// Mitsubishi GX Works2 project: PLC-Servo 실습 과제 1   PLC: Q03UDV

PROGRAM MAIN
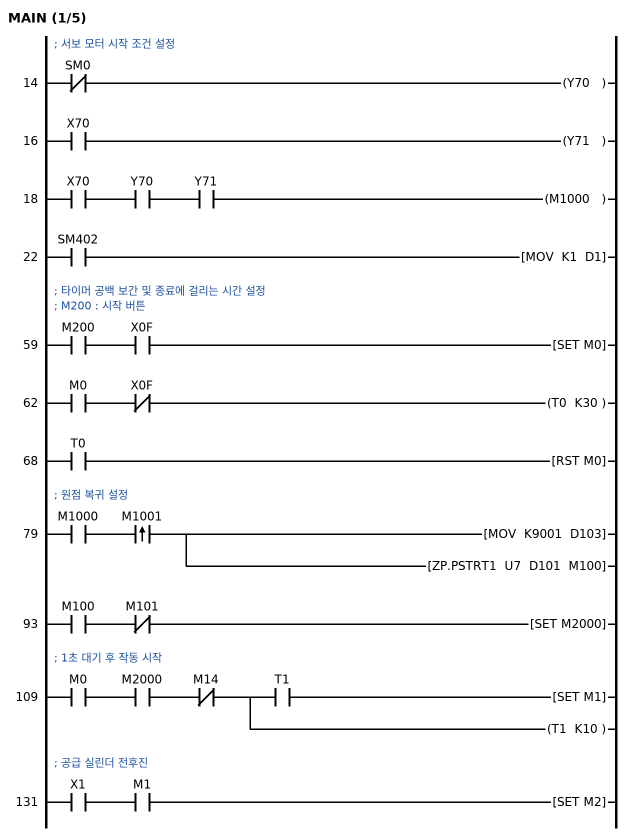
; 서보 모터 시작 조건 설정
14    LDI     SM0
      OUT     Y70
16    LD      X70
      OUT     Y71
18    LD      X70
      AND     Y70
      AND     Y71
      OUT     M1000
22    LD      SM402
      MOV     K1 D1
; 타이머 공백 보간 및 종료에 걸리는 시간 설정
; M200 : 시작 버튼
59    LD      M200
      AND     X0F
      SET     M0
62    LD      M0
      ANI     X0F
      OUT     T0 K30
68    LD      T0
      RST     M0
; 원점 복귀 설정
79    LD      M1000
      ANDP    M1001
      MOV     K9001 D103
      ZP.PSTRT1 U7 D101 M100
93    LD      M100
      ANI     M101
      SET     M2000
; 1초 대기 후 작동 시작
109   LD      M0
      AND     M2000
      ANI     M14
      MPS
      AND     T1
      SET     M1
      MPP
      OUT     T1 K10
; 공급 실린더 전후진
131   LD      X1
      AND     M1
      SET     M2
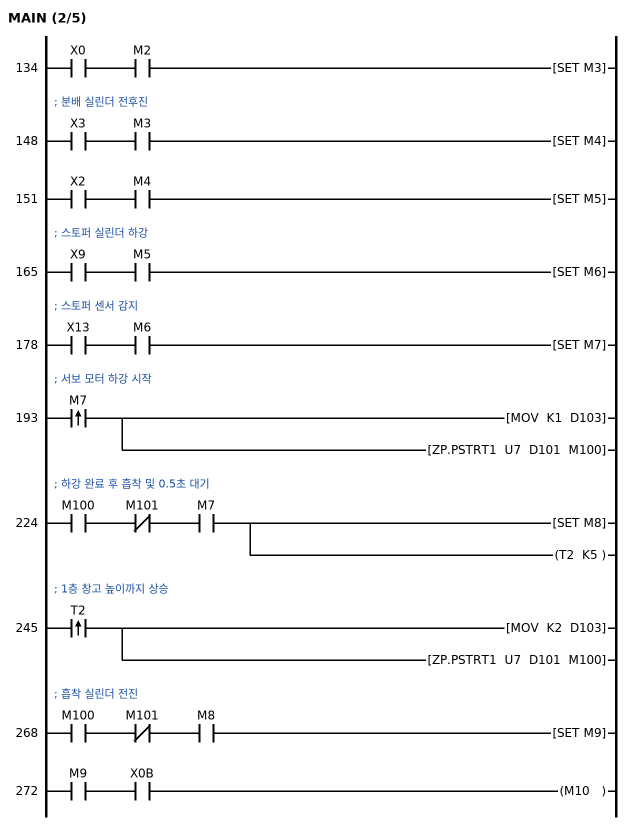
134   LD      X0
      AND     M2
      SET     M3
; 분배 실린더 전후진
148   LD      X3
      AND     M3
      SET     M4
151   LD      X2
      AND     M4
      SET     M5
; 스토퍼 실린더 하강
165   LD      X9
      AND     M5
      SET     M6
; 스토퍼 센서 감지
178   LD      X13
      AND     M6
      SET     M7
; 서보 모터 하강 시작
193   LDP     M7
      MOV     K1 D103
      ZP.PSTRT1 U7 D101 M100
; 하강 완료 후 흡착 및 0.5초 대기
224   LD      M100
      ANI     M101
      AND     M7
      SET     M8
      OUT     T2 K5
; 1층 창고 높이까지 상승
245   LDP     T2
      MOV     K2 D103
      ZP.PSTRT1 U7 D101 M100
; 흡착 실린더 전진
268   LD      M100
      ANI     M101
      AND     M8
      SET     M9
272   LD      M9
      AND     X0B
      OUT     M10
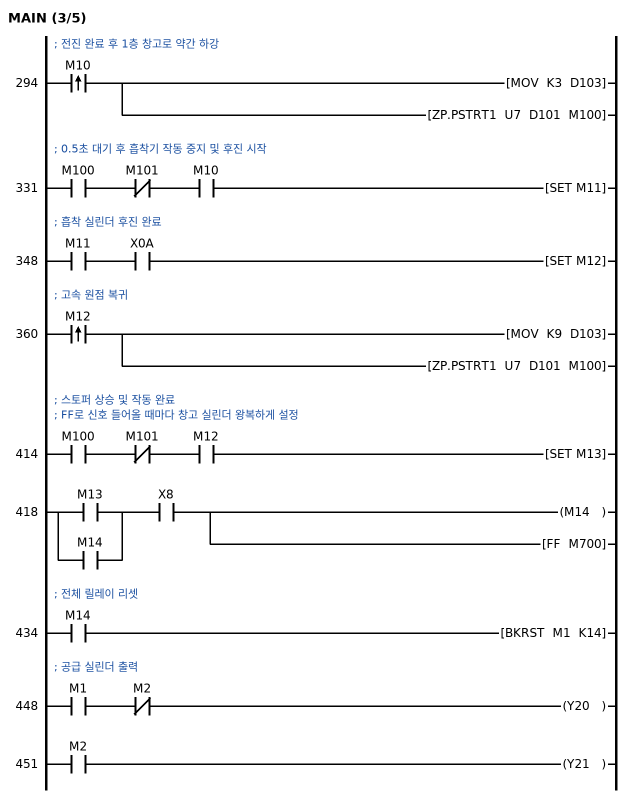
; 전진 완료 후 1층 창고로 약간 하강
294   LDP     M10
      MOV     K3 D103
      ZP.PSTRT1 U7 D101 M100
; 0.5초 대기 후 흡착기 작동 중지 및 후진 시작
331   LD      M100
      ANI     M101
      AND     M10
      SET     M11
; 흡착 실린더 후진 완료
348   LD      M11
      AND     X0A
      SET     M12
; 고속 원점 복귀
360   LDP     M12
      MOV     K9 D103
      ZP.PSTRT1 U7 D101 M100
; 스토퍼 상승 및 작동 완료
; FF로 신호 들어올 때마다 창고 실린더 왕복하게 설정
414   LD      M100
      ANI     M101
      AND     M12
      SET     M13
418   LD      M13
      OR      M14
      AND     X8
      OUT     M14
      FF      M700
; 전체 릴레이 리셋
434   LD      M14
      BKRST   M1 K14
; 공급 실린더 출력
448   LD      M1
      ANI     M2
      OUT     Y20
451   LD      M2
      OUT     Y21
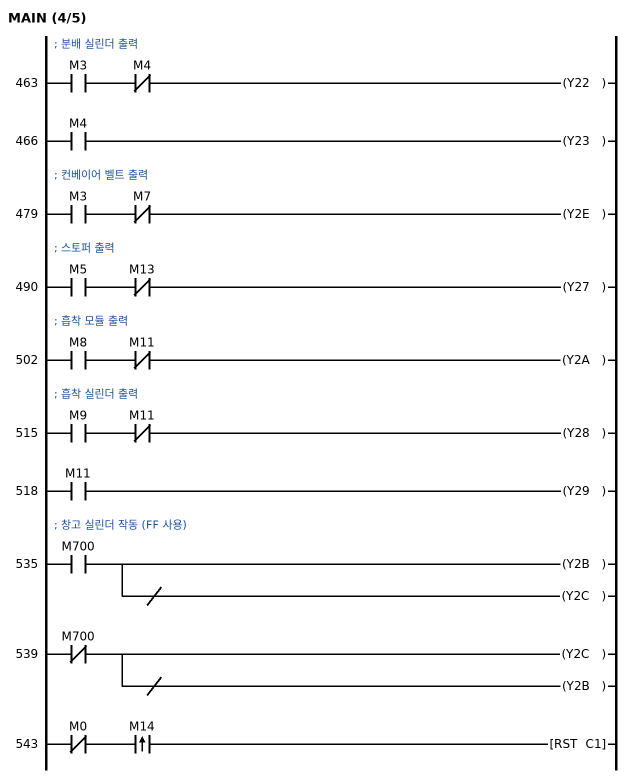
; 분배 실린더 출력
463   LD      M3
      ANI     M4
      OUT     Y22
466   LD      M4
      OUT     Y23
; 컨베이어 벨트 출력
479   LD      M3
      ANI     M7
      OUT     Y2E
; 스토퍼 출력
490   LD      M5
      ANI     M13
      OUT     Y27
; 흡착 모듈 출력
502   LD      M8
      ANI     M11
      OUT     Y2A
; 흡착 실린더 출력
515   LD      M9
      ANI     M11
      OUT     Y28
518   LD      M11
      OUT     Y29
; 창고 실린더 작동 (FF 사용)
535   LD      M700
      OUT     Y2B
      INV
      OUT     Y2C
539   LDI     M700
      OUT     Y2C
      INV
      OUT     Y2B
543   LDI     M0
      ANDP    M14
      RST     C1
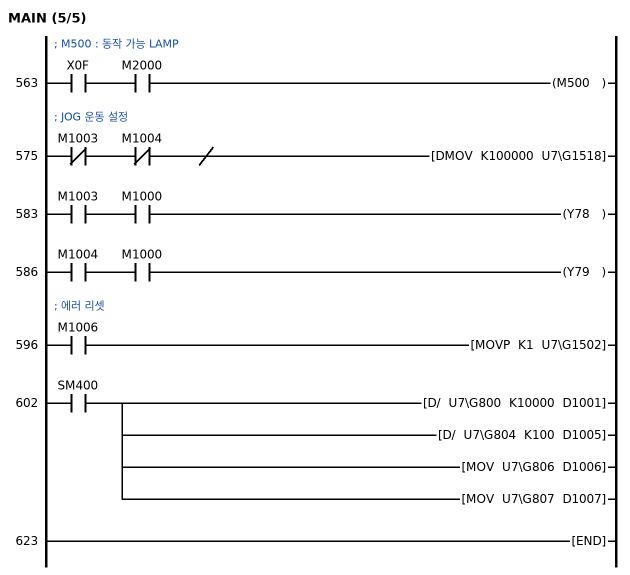
; M500 : 동작 가능 LAMP
563   LD      X0F
      AND     M2000
      OUT     M500
; JOG 운동 설정
575   LDI     M1003
      ANI     M1004
      INV
      DMOV    K100000 U7\G1518
583   LD      M1003
      AND     M1000
      OUT     Y78
586   LD      M1004
      AND     M1000
      OUT     Y79
; 에러 리셋
596   LD      M1006
      MOVP    K1 U7\G1502
602   LD      SM400
      D/      U7\G800 K10000 D1001
      D/      U7\G804 K100 D1005
      MOV     U7\G806 D1006
      MOV     U7\G807 D1007
623   END
END_PROGRAM
